(* CODESYS project ReflectiveSensor.xml

Project tree, tasks and I/O mapping:
  function block ReflectiveSensor [LD]
*)

// ReflectiveSensor
FUNCTION_BLOCK ReflectiveSensor
// The reflective sensor function block represents retro-reflective sensor functionality. 
// When the sensor no longer sees its reflection (meaning it is blocked) this function block will output to Q after the OnDelay time has passed,
// and will continue to output until the sensor sees its reflection again (meaning it is unblocked), AND the OffDelay time has passed.
VAR_INPUT
	IN: 				BOOL;				//
	OnDelay: 			TIME;				//
	OffDelay: 			TIME;				//
END_VAR
VAR_OUTPUT
	Q: 					BOOL;				//
END_VAR
VAR
	_OnDelayTimer: 		TON;				//
	_OffDelayTimer: 	TON;				//
END_VAR

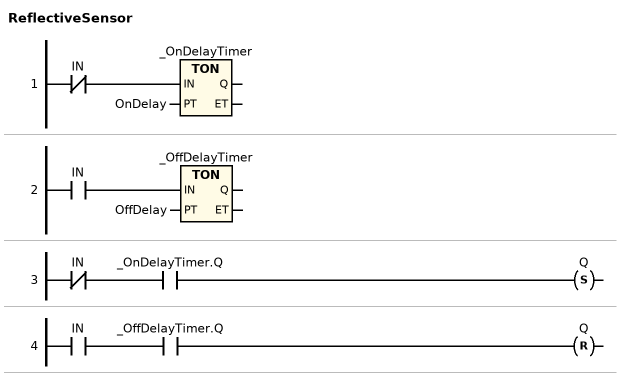
// NETWORK 1
_OnDelayTimer(IN := NOT IN, PT := OnDelay); // TON

// NETWORK 2
_OffDelayTimer(IN := IN, PT := OffDelay); // TON

// NETWORK 3
Q S= NOT IN AND _OnDelayTimer.Q;

// NETWORK 4
Q R= IN AND _OffDelayTimer.Q;

END_FUNCTION_BLOCK
